{attribute 'no_explicit_call' := 'DigitalInputNC is a class, do not call this POU directly, use a method'}
{attribute 'hide_all_locals'}
FUNCTION_BLOCK DigitalInputNC EXTENDS base IMPLEMENTS I_DigitalInput
VAR
    _input   AT %I* : BOOL;
    _signal  : BoolForceable(concat(name, ' forceable'), GVL_Logger.Logger);
END_VAR

METHOD FB_Init : BOOL
VAR_INPUT
    bInitRetains : BOOL;
    bInCopyCode  : BOOL;
    name         : STRING;
    logger       : I_Logger;
END_VAR
_signal.bind(_input);
END_METHOD

PROPERTY isActive : bool
GET
isActive := NOT _signal.value;
END_GET
END_PROPERTY

PROPERTY isNotActive : bool
GET
isNotActive := _signal.value;
END_GET
END_PROPERTY

PROPERTY signal : I_ForceableBOOL
GET
signal := _signal;
END_GET
END_PROPERTY

END_FUNCTION_BLOCK

(* stored: Version 1.1.0.1, ProductVersion 3.1.4026.18
   POU DigitalInputNC: Id {715fc0cf-2eef-43dc-af49-dd73af17a4b8}, SpecialFunc None
   Method FB_Init: Id {12345678-abcd-ef01-2345-6789abcdef01}
   Property isActive: Id {7096b06f-4d23-4173-9a0e-2d8432d559db}
   Get Get: Id {130ccbce-e396-44ac-9c45-da6e6a9fe1b0}
   Property isNotActive: Id {c22a03c0-d059-4087-b358-59756c84e8ea}
   Get Get: Id {88ea4f36-d219-4787-8089-a5a753182e06}
   Property signal: Id {11223344-5566-7788-99aa-bbccddeeff00}
   Get Get: Id {22334455-6677-8899-aabb-ccddeeff0011} *)
